// TIA Portal project "stokarabasifinal" (V16)

(* hardware
DEVICE "S7-1200 station_1"  S7-1200 Station
   slot 0: "Rack_0"  S7-1200 Rack  Rack  V1.0
   slot 1: "PLC_1"  CPU 1214C DC/DC/DC  6ES7 214-1AE30-0XB0  V2.2
*)

// ===== PLC "PLC_1"  CPU 1214C DC/DC/DC =====

VAR_GLOBAL   // PLC tag table "Default tag table"
   "LS_STOP1" AT %I0.0 : Bool;
   "LS_SLOW1" AT %I0.1 : Bool;
   "LS_SLOW2" AT %I0.2 : Bool;
   "LS_STOP2" AT %I0.3 : Bool;
   "MANUAL/AUTOMATIC" AT %I0.4 : Bool;
   "ACİL STOP" AT %I0.5 : Bool;
   "YUKARI START" AT %I0.6 : Bool;
   "AŞAĞI START" AT %I0.7 : Bool;
   "TERMİK" AT %I1.0 : Bool;
   "YUKARI YÖN" AT %Q0.0 : Bool;
   "AŞAĞI YÖN" AT %Q0.1 : Bool;
   "MOTOR SLOW" AT %Q0.2 : Bool;
   "MOTOR FAST_1" AT %Q0.3 : Bool;
   "MOTOR FAST_2" AT %Q0.4 : Bool;
   "YUKARI OTOMATİK" AT %M10.0 : Bool;
   "AŞAĞI OTOMATİK" AT %M10.1 : Bool;
   "YUKARI MANUAL" AT %M10.2 : Bool;
   "AŞAĞI MANUAL" AT %M10.3 : Bool;
   "AŞAĞI YON MARKERİ" AT %M10.4 : Bool;
   "YUKARI YON MARKERİ" AT %M10.5 : Bool;
   "HZ1 MARKERİ" AT %M10.6 : Bool;
   "HZ2 MARKERİ" AT %M10.7 : Bool;
   "FAULT LAMP" AT %Q0.5 : Bool;
   "ARIZA MARKERİ" AT %M11.0 : Bool;
   "Tag_1" AT %M60.0 : Bool;
   "Tag_2" AT %M60.1 : Bool;
   "Tag_3" AT %M60.2 : Bool;
   "Tag_4" AT %M60.3 : Bool;
   "Tag_6" AT %M60.5 : Bool;
   "Tag_5" AT %M60.4 : Bool;
   "Tag_7" AT %M60.6 : Bool;
   "Tag_8" AT %M60.7 : Bool;
END_VAR

ORGANIZATION_BLOCK "Main"   // OB1, LAD, ProgramCycle
TITLE = "Main Program Sweep (Cycle)"
{ S7_Optimized_Access := 'TRUE' }
VERSION : 0.1
   VAR_TEMP   // added for the SCL form of the ladder/FBD networks
      _w1 : Bool;
      _w2 : Bool;
      _w3 : Bool;
      _w4 : Bool;
   END_VAR
BEGIN

REGION Network 1: YUKARI OTOMATİK ÇALIŞMA MARKERİ
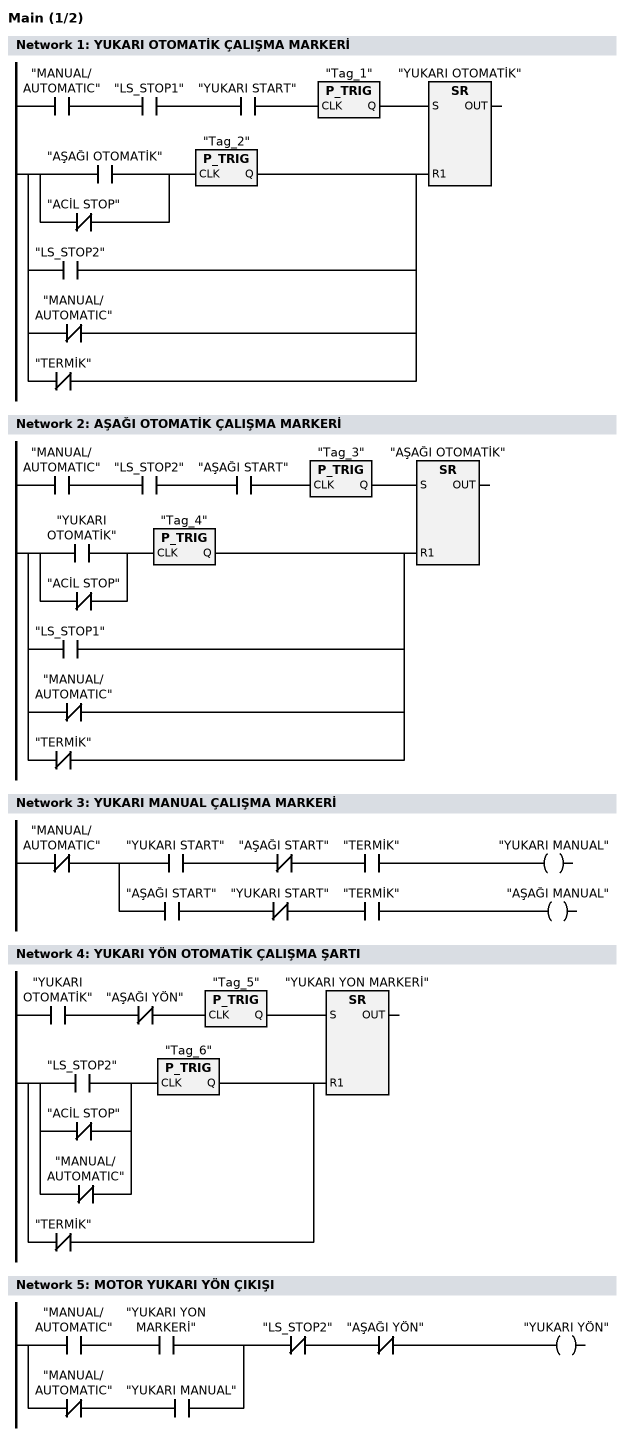
   RUNG wire#powerrail
      Contact( "MANUAL/AUTOMATIC" )
      Contact( "LS_STOP1" )
      Contact( "YUKARI START" )
      P_Trig( "Tag_1" )
      S_SR(operand := "YUKARI OTOMATİK", r1 := wire#w2)
   END_RUNG
   RUNG wire#powerrail
      Contact( "AŞAĞI OTOMATİK" )
      wire#w1
      P_Trig( "Tag_2" )
   END_RUNG wire#w2
   RUNG wire#powerrail
      I_Contact( "ACİL STOP" )
   END_RUNG wire#w1
   RUNG wire#powerrail
      Contact( "LS_STOP2" )
   END_RUNG wire#w2
   RUNG wire#powerrail
      I_Contact( "MANUAL/AUTOMATIC" )
   END_RUNG wire#w2
   RUNG wire#powerrail
      I_Contact( "TERMİK" )
   END_RUNG wire#w2
   // the same network as SCL:
   #_w1 := "MANUAL/AUTOMATIC" AND "LS_STOP1" AND "YUKARI START";
   #_w2 := #_w1 AND NOT "Tag_1";   // rising edge
   "Tag_1" := #_w1;
   #_w3 := "AŞAĞI OTOMATİK" OR NOT "ACİL STOP";
   #_w4 := #_w3 AND NOT "Tag_2";   // rising edge
   "Tag_2" := #_w3;
   IF #_w2 THEN
       "YUKARI OTOMATİK" := TRUE;   // SR flip-flop
   END_IF;
   IF #_w4 OR "LS_STOP2" OR NOT "MANUAL/AUTOMATIC" OR NOT "TERMİK" THEN "YUKARI OTOMATİK" := FALSE; END_IF;
END_REGION

REGION Network 2: AŞAĞI OTOMATİK ÇALIŞMA MARKERİ
   RUNG wire#powerrail
      Contact( "MANUAL/AUTOMATIC" )
      Contact( "LS_STOP2" )
      Contact( "AŞAĞI START" )
      P_Trig( "Tag_3" )
      S_SR(operand := "AŞAĞI OTOMATİK", r1 := wire#w2)
   END_RUNG
   RUNG wire#powerrail
      Contact( "YUKARI OTOMATİK" )
      wire#w1
      P_Trig( "Tag_4" )
   END_RUNG wire#w2
   RUNG wire#powerrail
      I_Contact( "ACİL STOP" )
   END_RUNG wire#w1
   RUNG wire#powerrail
      Contact( "LS_STOP1" )
   END_RUNG wire#w2
   RUNG wire#powerrail
      I_Contact( "MANUAL/AUTOMATIC" )
   END_RUNG wire#w2
   RUNG wire#powerrail
      I_Contact( "TERMİK" )
   END_RUNG wire#w2
   // the same network as SCL:
   #_w1 := "MANUAL/AUTOMATIC" AND "LS_STOP2" AND "AŞAĞI START";
   #_w2 := #_w1 AND NOT "Tag_3";   // rising edge
   "Tag_3" := #_w1;
   #_w3 := "YUKARI OTOMATİK" OR NOT "ACİL STOP";
   #_w4 := #_w3 AND NOT "Tag_4";   // rising edge
   "Tag_4" := #_w3;
   IF #_w2 THEN
       "AŞAĞI OTOMATİK" := TRUE;   // SR flip-flop
   END_IF;
   IF #_w4 OR "LS_STOP1" OR NOT "MANUAL/AUTOMATIC" OR NOT "TERMİK" THEN "AŞAĞI OTOMATİK" := FALSE; END_IF;
END_REGION

REGION Network 3: YUKARI MANUAL ÇALIŞMA MARKERİ
   RUNG wire#powerrail
      I_Contact( "MANUAL/AUTOMATIC" )
      wire#w1
      Contact( "YUKARI START" )
      I_Contact( "AŞAĞI START" )
      Contact( "TERMİK" )
      Coil( "YUKARI MANUAL" )
   END_RUNG
   RUNG wire#w1
      Contact( "AŞAĞI START" )
      I_Contact( "YUKARI START" )
      Contact( "TERMİK" )
      Coil( "AŞAĞI MANUAL" )
   END_RUNG
   // the same network as SCL:
   "YUKARI MANUAL" := NOT "MANUAL/AUTOMATIC" AND "YUKARI START" AND NOT "AŞAĞI START" AND "TERMİK";
   "AŞAĞI MANUAL" := NOT "MANUAL/AUTOMATIC" AND "AŞAĞI START" AND NOT "YUKARI START" AND "TERMİK";
END_REGION

REGION Network 4: YUKARI YÖN OTOMATİK ÇALIŞMA ŞARTI
   RUNG wire#powerrail
      Contact( "YUKARI OTOMATİK" )
      I_Contact( "AŞAĞI YÖN" )
      P_Trig( "Tag_5" )
      S_SR(operand := "YUKARI YON MARKERİ", r1 := wire#w2)
   END_RUNG
   RUNG wire#powerrail
      Contact( "LS_STOP2" )
      wire#w1
      P_Trig( "Tag_6" )
   END_RUNG wire#w2
   RUNG wire#powerrail
      I_Contact( "ACİL STOP" )
   END_RUNG wire#w1
   RUNG wire#powerrail
      I_Contact( "MANUAL/AUTOMATIC" )
   END_RUNG wire#w1
   RUNG wire#powerrail
      I_Contact( "TERMİK" )
   END_RUNG wire#w2
   // the same network as SCL:
   #_w1 := "YUKARI OTOMATİK" AND NOT "AŞAĞI YÖN";
   #_w2 := #_w1 AND NOT "Tag_5";   // rising edge
   "Tag_5" := #_w1;
   #_w3 := "LS_STOP2" OR NOT "ACİL STOP" OR NOT "MANUAL/AUTOMATIC";
   #_w4 := #_w3 AND NOT "Tag_6";   // rising edge
   "Tag_6" := #_w3;
   IF #_w2 THEN
       "YUKARI YON MARKERİ" := TRUE;   // SR flip-flop
   END_IF;
   IF #_w4 OR NOT "TERMİK" THEN "YUKARI YON MARKERİ" := FALSE; END_IF;
END_REGION

REGION Network 5: MOTOR YUKARI YÖN ÇIKIŞI
   RUNG wire#powerrail
      Contact( "MANUAL/AUTOMATIC" )
      Contact( "YUKARI YON MARKERİ" )
      wire#w1
      I_Contact( "LS_STOP2" )
      I_Contact( "AŞAĞI YÖN" )
      Coil( "YUKARI YÖN" )
   END_RUNG
   RUNG wire#powerrail
      I_Contact( "MANUAL/AUTOMATIC" )
      Contact( "YUKARI MANUAL" )
   END_RUNG wire#w1
   // the same network as SCL:
   "YUKARI YÖN" := (("MANUAL/AUTOMATIC" AND "YUKARI YON MARKERİ") OR (NOT "MANUAL/AUTOMATIC" AND "YUKARI MANUAL")) AND NOT "LS_STOP2" AND NOT "AŞAĞI YÖN";
END_REGION

REGION Network 6
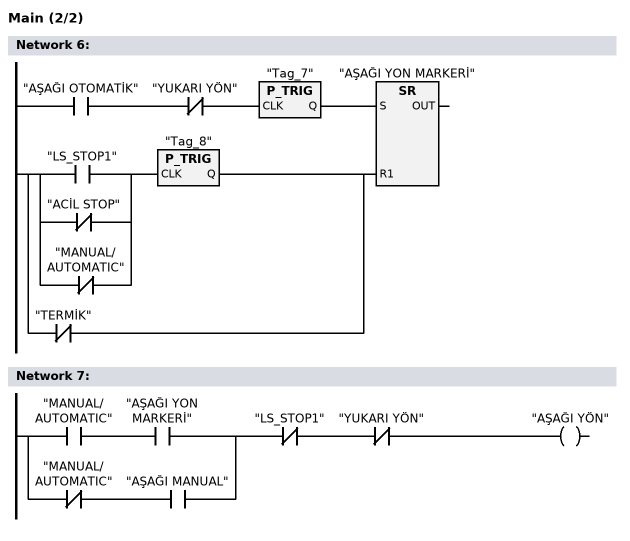
   RUNG wire#powerrail
      Contact( "AŞAĞI OTOMATİK" )
      I_Contact( "YUKARI YÖN" )
      P_Trig( "Tag_7" )
      S_SR(operand := "AŞAĞI YON MARKERİ", r1 := wire#w2)
   END_RUNG
   RUNG wire#powerrail
      Contact( "LS_STOP1" )
      wire#w1
      P_Trig( "Tag_8" )
   END_RUNG wire#w2
   RUNG wire#powerrail
      I_Contact( "ACİL STOP" )
   END_RUNG wire#w1
   RUNG wire#powerrail
      I_Contact( "MANUAL/AUTOMATIC" )
   END_RUNG wire#w1
   RUNG wire#powerrail
      I_Contact( "TERMİK" )
   END_RUNG wire#w2
   // the same network as SCL:
   #_w1 := "AŞAĞI OTOMATİK" AND NOT "YUKARI YÖN";
   #_w2 := #_w1 AND NOT "Tag_7";   // rising edge
   "Tag_7" := #_w1;
   #_w3 := "LS_STOP1" OR NOT "ACİL STOP" OR NOT "MANUAL/AUTOMATIC";
   #_w4 := #_w3 AND NOT "Tag_8";   // rising edge
   "Tag_8" := #_w3;
   IF #_w2 THEN
       "AŞAĞI YON MARKERİ" := TRUE;   // SR flip-flop
   END_IF;
   IF #_w4 OR NOT "TERMİK" THEN "AŞAĞI YON MARKERİ" := FALSE; END_IF;
END_REGION

REGION Network 7
   RUNG wire#powerrail
      Contact( "MANUAL/AUTOMATIC" )
      Contact( "AŞAĞI YON MARKERİ" )
      wire#w1
      I_Contact( "LS_STOP1" )
      I_Contact( "YUKARI YÖN" )
      Coil( "AŞAĞI YÖN" )
   END_RUNG
   RUNG wire#powerrail
      I_Contact( "MANUAL/AUTOMATIC" )
      Contact( "AŞAĞI MANUAL" )
   END_RUNG wire#w1
   // the same network as SCL:
   "AŞAĞI YÖN" := (("MANUAL/AUTOMATIC" AND "AŞAĞI YON MARKERİ") OR (NOT "MANUAL/AUTOMATIC" AND "AŞAĞI MANUAL")) AND NOT "LS_STOP1" AND NOT "YUKARI YÖN";
END_REGION
END_ORGANIZATION_BLOCK